FUNCTION_BLOCK State
VAR_INPUT
END_VAR
VAR_OUTPUT
END_VAR
VAR
END_VAR

METHOD Run : BOOL
VAR_INPUT
END_VAR
END_METHOD

METHOD Start : BOOL
VAR_INPUT
END_VAR
END_METHOD

METHOD Stop : BOOL
VAR_INPUT
END_VAR
END_METHOD

METHOD Transition : POINTER TO State
VAR_INPUT
END_VAR
Transition := ADR(THIS^);
END_METHOD

END_FUNCTION_BLOCK

(* stored: Version 1.1.0.1, ProductVersion 3.1.4024.3
   POU State: Id {9dbb020e-07f3-49c6-9250-91502d4b2d6f}, SpecialFunc None
   Method Run: Id {664c0116-4061-4da4-9554-8fa83562b818}
   Method Start: Id {2d8f2914-360e-48d1-b86f-5b084ae01727}
   Method Stop: Id {c35322c8-340e-4abf-9743-94423fed4e20}
   Method Transition: Id {f74520f1-202a-4ad8-9598-49eadd8359d5} *)
